// ===== Calibration Param SDO Hybrid Logic (startup-sequential, then on-demand) =====
// Sequential trigger (bCalibParamStep statemachine) is used at startup or force, otherwise parallel/on-demand.

FUNCTION_BLOCK FB_WriteCalibrationParameters
VAR_INPUT
    bEnable : BOOL;
END_VAR
VAR_IN_OUT
    stDS402Drive         : ST_DS402Drive;
    stMotionStage        : ST_MotionStage;
    stMCS2ChanParameter	: ST_MCS2ChanParameter;
END_VAR

VAR_OUTPUT
   bCalibrationsParamsSet : BOOL;
END_VAR
VAR
    {attribute 'hide'}
    fbSafeDirWrite              : FB_EcCoESdoWrite;
    {attribute 'hide'}
    fbChannelTypeWrite          : FB_EcCoESdoWrite;
    {attribute 'hide'}
    fbPositionerTypeWrite       : FB_EcCoESdoWrite;
    {attribute 'hide'}
    fbCalibrationOptWrite       : FB_EcCoESdoWrite;
    {attribute 'hide'}
    ftPositionerTypeSetDone     : F_TRIG;
    {attribute 'hide'}
    ftCalibrationOptSetDone     : F_TRIG;
    {attribute 'hide'}
    ftSafeDirSetDone            : F_TRIG;
    {attribute 'hide'}
    ftChannelTypeSetDone        : F_TRIG;
    {attribute 'hide'}
    nRecentPositionerType       : UDINT;
    {attribute 'hide'}
    nRecentCalibrationOpt       : UDINT;
    {attribute 'hide'}
    nRecentSafeDir              : BOOL;
    {attribute 'hide'}
    nRecentChannelType          : UDINT;
    tonStartUp : TON;
    nCalibParamStep : INT := 0; // 0: idle, 1~5: write steps, 10: done, -1: error
    bForceSequentialSDOs : BOOL := FALSE;
    bErrorAcknowledge: BOOL;
END_VAR

IF bEnable THEN
    tonStartUp(
        IN := bEnable AND NOT bCalibrationsParamsSet,
        PT := T#4S
    );

    IF (NOT tonStartUp.Q) AND (nCalibParamStep <> 0) AND (NOT bForceSequentialSDOs) THEN
        nCalibParamStep := 0;
    END_IF

    IF (nCalibParamStep = -1) AND bErrorAcknowledge THEN
        nCalibParamStep := 0;
        stMotionStage.bError := FALSE;
        stMotionStage.nErrorId := 0;
    END_IF

    ftCalibrationOptSetDone(CLK := fbCalibrationOptWrite.bBusy);

    IF tonStartUp.Q OR bForceSequentialSDOs THEN

        CASE nCalibParamStep OF
        0:
            bCalibrationsParamsSet := FALSE;
            fbCalibrationOptWrite.bExecute := FALSE;
            nCalibParamStep := 1;

        1:
            IF (stMCS2ChanParameter.nCalibrationOpt <> nRecentCalibrationOpt) THEN
                fbCalibrationOptWrite.bExecute := TRUE;
                IF ftCalibrationOptSetDone.Q THEN
                    IF fbCalibrationOptWrite.bError THEN
                        stMotionStage.bError := fbCalibrationOptWrite.bError;
                        stMotionStage.nErrorId := fbCalibrationOptWrite.nErrId;
                        nCalibParamStep := -1;
                    ELSE
                        nRecentCalibrationOpt := stMCS2ChanParameter.nCalibrationOpt;
                        fbCalibrationOptWrite.bExecute := FALSE;
                        nCalibParamStep := 10;
                    END_IF
                END_IF
            ELSE
                nCalibParamStep := 10;
            END_IF

        10:
            bCalibrationsParamsSet := TRUE;
        -1:
            bCalibrationsParamsSet := FALSE;
        ELSE
            nCalibParamStep := 0;
        END_CASE
    ELSE
        fbCalibrationOptWrite.bExecute := (stMCS2ChanParameter.nCalibrationOpt <> nRecentCalibrationOpt);

        IF ftCalibrationOptSetDone.Q THEN
            IF fbCalibrationOptWrite.bError THEN
                stMotionStage.bError := fbCalibrationOptWrite.bError;
                stMotionStage.nErrorId := fbCalibrationOptWrite.nErrId;
            ELSE
                nRecentCalibrationOpt := stMCS2ChanParameter.nCalibrationOpt;
                bCalibrationsParamsSet := TRUE;
            END_IF
            fbCalibrationOptWrite.bExecute := FALSE;
        END_IF
    END_IF

    fbCalibrationOptWrite(
        sNetId     := stMotionStage.stAxisParameters.sAmsNetId,
        nSlaveAddr := stDS402Drive.nSlaveAddr,
        nIndex     := stMCS2ChanParameter.nChanCalibrationOptIdx,
        nSubIndex  := 0,
        pSrcBuf    := ADR(stMCS2ChanParameter.nCalibrationOpt),
        cbBufLen   := SIZEOF(stMCS2ChanParameter.nCalibrationOpt)
    );

    bCalibrationsParamsSet R= fbCalibrationOptWrite.bBusy;
END_IF

END_FUNCTION_BLOCK

(* stored: Version 1.1.0.1
   POU FB_WriteCalibrationParameters: Id {6f8141b3-3a18-4ecd-8d0f-d7b01f6561a0}, SpecialFunc None *)
